(* IEC 61131-3 sources: twincat-conveyor-simulator/PLC, 2 files *)

(* ---- FB_Conveyor.st ---- *)
FUNCTION_BLOCK FB_Conveyor
VAR_INPUT
    bStart          : BOOL;
    bStop           : BOOL;
    bReset          : BOOL;
    bEmergencyStop  : BOOL;
    bPartSensor     : BOOL;
END_VAR
VAR_OUTPUT
    bMotorRunning   : BOOL;
    bFaultActive    : BOOL;
    nPartCount      : UDINT;
    eState          : E_MachineState;
END_VAR
VAR
    rPartSensor     : R_TRIG;
END_VAR

IF bEmergencyStop THEN
    bFaultActive := TRUE;
    bMotorRunning := FALSE;
    eState := E_MachineState.Faulted;
ELSIF bReset THEN
    bFaultActive := FALSE;
    bMotorRunning := FALSE;
    nPartCount := 0;
    eState := E_MachineState.Stopped;
ELSE
    CASE eState OF
        E_MachineState.Stopped:
            bMotorRunning := FALSE;
            IF bStart AND NOT bFaultActive THEN
                bMotorRunning := TRUE;
                eState := E_MachineState.Running;
            END_IF
        E_MachineState.Running:
            bMotorRunning := TRUE;
            IF bStop THEN
                bMotorRunning := FALSE;
                eState := E_MachineState.Stopped;
            END_IF
        E_MachineState.Faulted:
            bMotorRunning := FALSE;
    ELSE
        bMotorRunning := FALSE;
        eState := E_MachineState.Stopped;
    END_CASE
END_IF

rPartSensor(CLK := bPartSensor);
IF rPartSensor.Q AND bMotorRunning THEN
    nPartCount := nPartCount + 1;
END_IF

(* ---- MAIN.st ---- *)
PROGRAM MAIN
VAR
    fbConveyor     : FB_Conveyor;
    tonPartPulse   : TON;
    bSimulatedPart : BOOL;
END_VAR

IF GVL_HMI.bAutoSimulatePart AND GVL_HMI.bMotorRunning THEN
    tonPartPulse(IN := NOT tonPartPulse.Q, PT := T#3S);
    bSimulatedPart := tonPartPulse.ET >= T#2500MS;
ELSE
    tonPartPulse(IN := FALSE, PT := T#3S);
    bSimulatedPart := FALSE;
END_IF

GVL_HMI.bPartSensor := bSimulatedPart OR GVL_HMI.bManualPartSensor;

fbConveyor(
    bStart         := GVL_HMI.bStartCommand,
    bStop          := GVL_HMI.bStopCommand,
    bReset         := GVL_HMI.bResetCommand,
    bEmergencyStop := GVL_HMI.bEmergencyStop,
    bPartSensor    := GVL_HMI.bPartSensor
);

GVL_HMI.bMotorRunning := fbConveyor.bMotorRunning;
GVL_HMI.bFaultActive  := fbConveyor.bFaultActive;
GVL_HMI.nPartCount    := fbConveyor.nPartCount;
GVL_HMI.eMachineState := fbConveyor.eState;

GVL_HMI.bStartCommand := FALSE;
GVL_HMI.bStopCommand  := FALSE;
GVL_HMI.bResetCommand := FALSE;
